FUNCTION F_MoveTU_DataIndexEmulation : DINT
(**************************************************************************************
 * 	Application		:	BoxControl Framework
 *	Revision		:	$Revision: 404529 $
 *	Revision date	:	$Date: 2018-04-23 08:21:38 +0200 (Mo., 23 Apr 2018) $
 *	Last changed by	:	$Author: b7bolm $
 *	URL				:	$URL: http://almscdc.swisslog.com/repo/SWPD/Development/BoxControlFramework/20_Release/trunk/01_Software/BCF/BCF/JumpStart/20_Product/11_Emu/12_E_Functions/10_Lib/10_Conv/10_Functions/F_MoveTU_DataIndexEmulation.TcPOU $
 *
 *	Purpose			:	Moves TU data from a position.
 *
 * ------------------------------------------------------------------------------------
 *	Copyright Swisslog [IP AG], Switzerland. All rights reserved.
 * 
 * ------------------------------------------------------------------------------------
 *	
 * 	Revision History: 
 *
 * 	VERSION			DATE			INITIALS			DESCRIPTION
 *	0.1				01.01.2001		swl					Example
 *
 **************************************************************************************)
VAR_INPUT
	eFunctionNumber	: E_FunctionNumber; // Function number of corresponding function
	mZoneNumber 	: INT; // Zone number
END_VAR

VAR
	STI_Instance		: ITF_SubsystemTransportEmulation; // Instance to compare valid interfaces
	eFunctionNumberSTI : E_FunctionNumber;
END_VAR

// Check if function number is valid
IF eFunctionNumber > E_FunctionNumber.F_BEGIN_FUNCTION AND
   eFunctionNumber < E_FunctionNumber.F_END_FUNCTION THEN
  
	// Check reference is valid
	IF __ISVALIDREF(FunctionRegistryEmulation[eFunctionNumber].rFunction) THEN
   		// Return tu data index
   		F_MoveTU_DataIndexEmulation := FunctionRegistryEmulation[eFunctionNumber].rFunction.M_MoveTU_DataIndex(mZoneNumber := mZoneNumber);
	END_IF
	
ELSIF eFunctionNumber > E_FunctionNumber.F_BEGIN_EXTERN_FUNCTION AND
	  eFunctionNumber < E_FunctionNumber.F_END_EXTERN_FUNCTION THEN

	// Return tu data index
	IF __QUERYINTERFACE(fbSTI_ChannelsEmulation[eFunctionNumber].Instance,STI_Instance) THEN
		// Return tu data index
		F_MoveTU_DataIndexEmulation := fbSTI_ChannelsEmulation[eFunctionNumber].Instance.M_MoveTU_DataIndex();
	END_IF
END_IF

END_FUNCTION

(* stored: Version 1.1.0.1, ProductVersion 3.1.4022.12
   POU F_MoveTU_DataIndexEmulation: Id {1ec0c8ea-2540-4e58-b1b7-90a777b360d3}, SpecialFunc None *)
